// SIMATIC STEP 7 (V5.x) project Stend2
// CPU: CPU 315-2 DP
// station: P_ADR_BUS
// station: Hardware
// station: SIMATIC 300(1)
// program: S7 Program(3)

SYMBOL_TABLE
"Koncevik"	I 4.1	BOOL
"Induct sensor"	I 5.0	BOOL
END_SYMBOL_TABLE

FUNCTION_BLOCK FB 1
VERSION : 0.1
BEGIN
// (block stored without names or comments; labels and parameter names are numbered)
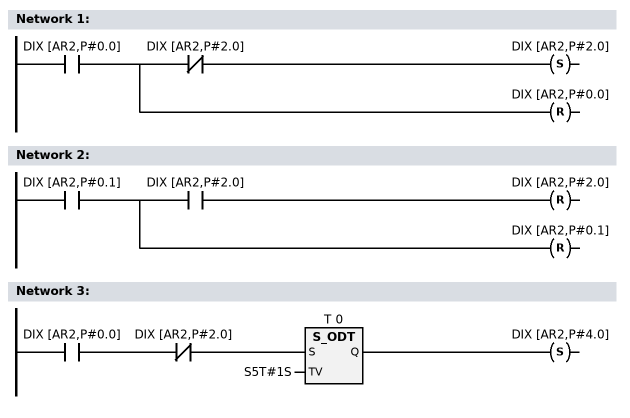
NETWORK
TITLE =
      A     DIX [AR2,P#0.0];
      =     L 0.0;
      A     L 0.0;
      AN    DIX [AR2,P#2.0];
      S     DIX [AR2,P#2.0];
      A     L 0.0;
      BLD   102;
      R     DIX [AR2,P#0.0];
NETWORK
TITLE =
      A     DIX [AR2,P#0.1];
      =     L 0.0;
      A     L 0.0;
      A     DIX [AR2,P#2.0];
      R     DIX [AR2,P#2.0];
      A     L 0.0;
      BLD   102;
      R     DIX [AR2,P#0.1];
NETWORK
TITLE =
      A     DIX [AR2,P#0.0];
      AN    DIX [AR2,P#2.0];
      L     S5T#1S;
      SD    T 0;
      NOP   0;
      NOP   0;
      NOP   0;
      A     T 0;
      S     DIX [AR2,P#4.0];
END_FUNCTION_BLOCK

// FB 41: know-how protected block, not included

FUNCTION FC 5 : VOID
VERSION : 0.1
BEGIN
// (block stored without names or comments; labels and parameter names are numbered)
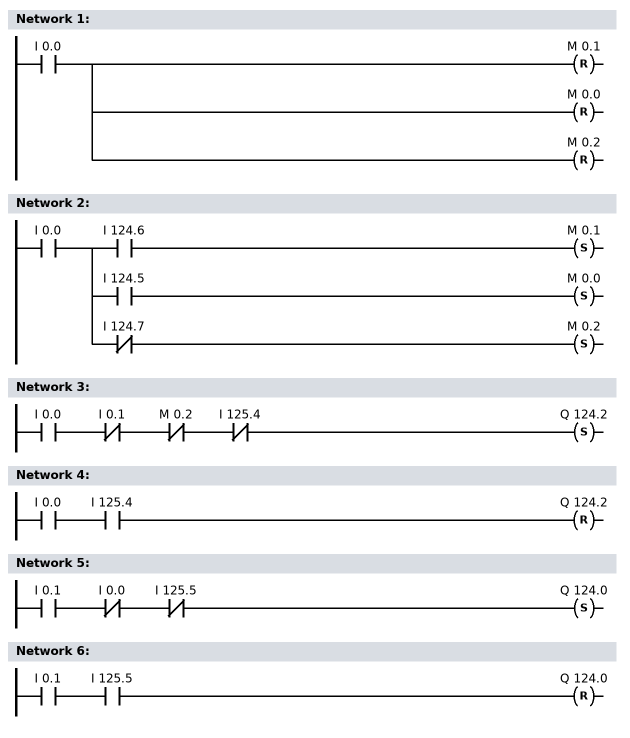
NETWORK
TITLE =
      A     I 0.0;
      R     M 0.1;
      R     M 0.0;
      R     M 0.2;
NETWORK
TITLE =
      A     I 0.0;
      =     L 0.0;
      A     L 0.0;
      A     I 124.6;
      S     M 0.1;
      A     L 0.0;
      A     I 124.5;
      S     M 0.0;
      A     L 0.0;
      AN    I 124.7;
      S     M 0.2;
NETWORK
TITLE =
      A     I 0.0;
      AN    I 0.1;
      AN    M 0.2;
      AN    I 125.4;
      S     Q 124.2;
NETWORK
TITLE =
      A     I 0.0;
      A     I 125.4;
      R     Q 124.2;
NETWORK
TITLE =
      A     I 0.1;
      AN    I 0.0;
      AN    I 125.5;
      S     Q 124.0;
NETWORK
TITLE =
      A     I 0.1;
      A     I 125.5;
      R     Q 124.0;
END_FUNCTION

FUNCTION FC 11 : VOID
VERSION : 0.1
BEGIN
// (block stored without names or comments; labels and parameter names are numbered)
NETWORK
TITLE =
NETWORK
TITLE =
      CALL  FC 7 (
           $1                       := #PARAM1,
           $2                       := L#968728430,
           $3                       := L#0,
           $4                       := 32512,
           $5                       := 27649,
           $6                       := -1,
           $7                       := -8865,
           $8                       := #PARAM2,
           $9                       := #PARAM3,
           $10                      := #PARAM4);
END_FUNCTION

// FC 106: know-how protected block, not included

DATA_BLOCK DB 1
VERSION : 0.1
BEGIN
// 4 bytes; values not shown
END_DATA_BLOCK

DATA_BLOCK DB 2
VERSION : 0.1
BEGIN
// 4 bytes; values not shown
END_DATA_BLOCK

DATA_BLOCK DB 3
VERSION : 0.1
BEGIN
// 4 bytes; values not shown
END_DATA_BLOCK

DATA_BLOCK DB 301
VERSION : 0.1
BEGIN
// 16 bytes; values not shown
END_DATA_BLOCK

ORGANIZATION_BLOCK OB 1
TITLE = Test
//Test
//
VERSION : 0.1
VAR_TEMP
  TEMP0 : BYTE ;
  TEMP1 : BYTE ;
  TEMP2 : BYTE ;
  TEMP3 : BYTE ;
  TEMP4 : BYTE ;
  TEMP5 : BYTE ;
  TEMP6 : INT ;
  TEMP7 : INT ;
  TEMP8 : INT ;
  TEMP9 : DATE_AND_TIME ;
END_VAR
BEGIN
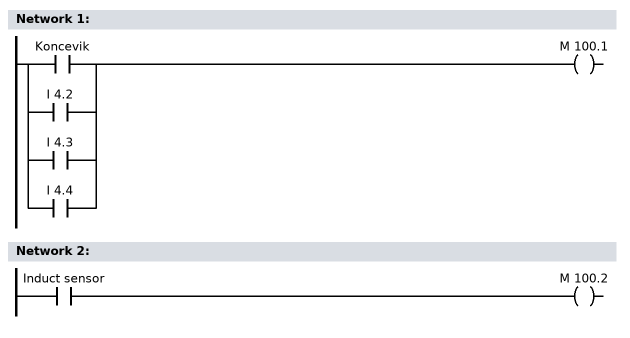
NETWORK
TITLE =
      O     "Koncevik";
      O     I 4.2;
      O     I 4.3;
      O     I 4.4;
      =     M 100.1;
NETWORK
TITLE =
      A     "Induct sensor";
      =     M 100.2;
END_ORGANIZATION_BLOCK

ORGANIZATION_BLOCK OB 80
VERSION : 0.1
BEGIN
// (block stored without names or comments; labels and parameter names are numbered)
END_ORGANIZATION_BLOCK

ORGANIZATION_BLOCK OB 86
VERSION : 0.1
BEGIN
// (block stored without names or comments; labels and parameter names are numbered)
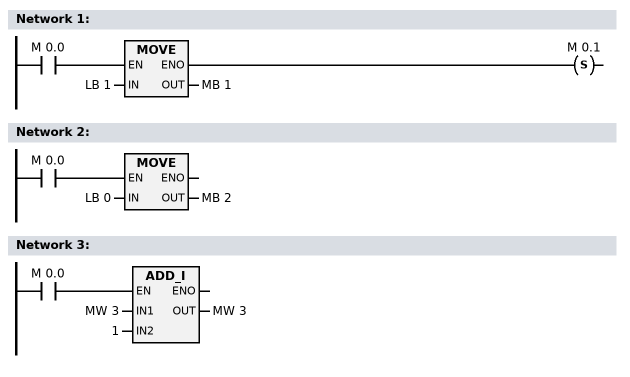
NETWORK
TITLE =
      A     M 0.0;
      JNB   M001;
      L     LB 1;
      T     MB 1;
      SET;
      SAVE;
      CLR;
M001: A     BR;
      S     M 0.1;
NETWORK
TITLE =
      A     M 0.0;
      JNB   M002;
      L     LB 0;
      T     MB 2;
M002: NOP   0;
NETWORK
TITLE =
      A     M 0.0;
      JNB   M003;
      L     MW 3;
      L     1;
      +I;
      T     MW 3;
M003: NOP   0;
END_ORGANIZATION_BLOCK
